// TIA Portal V17 export
FUNCTION "变频器通讯故障" : Void   // FC, LAD
{ S7_Optimized_Access := 'TRUE' }
VERSION : 0.1
// stored: AutoNumber true, IsIECCheckEnabled false, IsRetainMemResEnabled false, MemoryReserve 100, SetENOAutomatically false, UDAEnableTagReadback false
   VAR_TEMP   // added for the SCL form of the ladder/FBD networks
      _w1 : Bool;
   END_VAR
BEGIN

REGION Network 1: 变频器读取失败上升沿置位故障标志
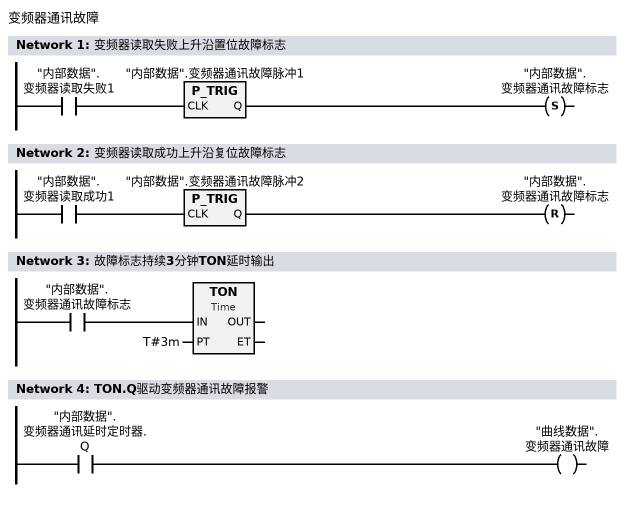
   RUNG wire#powerrail
      Contact( "内部数据".变频器读取失败1 )
      P_Trig( "内部数据".变频器通讯故障脉冲1 )
      S_Coil( "内部数据".变频器通讯故障标志 )
   END_RUNG
   // the same network as SCL:
   #_w1 := "内部数据".变频器读取失败1 AND NOT "内部数据".变频器通讯故障脉冲1;   // rising edge
   "内部数据".变频器通讯故障脉冲1 := "内部数据".变频器读取失败1;
   IF #_w1 THEN "内部数据".变频器通讯故障标志 := TRUE; END_IF;
END_REGION

REGION Network 2: 变频器读取成功上升沿复位故障标志
   RUNG wire#powerrail
      Contact( "内部数据".变频器读取成功1 )
      P_Trig( "内部数据".变频器通讯故障脉冲2 )
      R_Coil( "内部数据".变频器通讯故障标志 )
   END_RUNG
   // the same network as SCL:
   #_w1 := "内部数据".变频器读取成功1 AND NOT "内部数据".变频器通讯故障脉冲2;   // rising edge
   "内部数据".变频器通讯故障脉冲2 := "内部数据".变频器读取成功1;
   IF #_w1 THEN "内部数据".变频器通讯故障标志 := FALSE; END_IF;
END_REGION

REGION Network 3: 故障标志持续3分钟TON延时输出
   RUNG wire#powerrail
      Contact( "内部数据".变频器通讯故障标志 )
      { S7_Templates := "time_type := Time" } TON(pt := T#3m, et =>)
   END_RUNG
   // the same network as SCL:
   TON(IN := "内部数据".变频器通讯故障标志, PT := T#3m);
END_REGION

REGION Network 4: TON.Q驱动变频器通讯故障报警
   RUNG wire#powerrail
      Contact( "内部数据".变频器通讯延时定时器.Q )
      Coil( "曲线数据".变频器通讯故障 )
   END_RUNG
   // the same network as SCL:
   "曲线数据".变频器通讯故障 := "内部数据".变频器通讯延时定时器.Q;
END_REGION
END_FUNCTION
